{attribute 'GeneratedUsingTerminal: KL8519'}
{attribute addProperty BoxType "KL8519"}
{attribute addProperty Id "Channel_1AT %Q*Channel_D13646E30"}
{attribute addProperty CRC "2352243983"}
{attribute addProperty Size "0"}
TYPE KL8519_8C34650F :
STRUCT
	{attribute addProperty Name "Channel_1"}
	Channel_1 : Channel_D13646E3;
END_STRUCT
END_TYPE
